# EPICS substitutions: ek9000App/Db/EL1004.substitutions
file EL1004.template
{       pattern
        {
                TERMINAL,

        }
        {
        }
}
